PROGRAM MAIN
VAR
	TestSuite : T_TestSuite;
END_VAR

TestSuite.RunTests();

END_PROGRAM

(* stored: Version 1.1.0.1, ProductVersion 3.1.4024.15
   POU MAIN: Id {44005d96-5425-4ff5-9844-0eaf592c14f6}, SpecialFunc None *)
